Staubli VAL3: OpenPince_test.pgx

program OpenPince_test()
begin

  userPage(sEcran)
  cls(sEcran)

  close(tTool)
  open(tTool)
    put(sEcran, "Operation réalisé")
end
